FUNCTION_BLOCK Robotino (* Basic Function Block Type *)
  (* Standard: 61499-2 *)
  (* Version 0.0, 18/10/2022, Pranay Jhunjhunwala, Schneider Electric, Template *)
  PACKAGE Main;
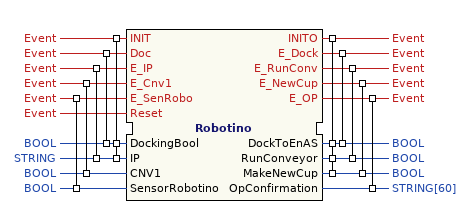
  EVENT_INPUT
    INIT WITH DockingBool, IP; (* Initialization Request *)
    Doc WITH DockingBool; (* Normal Execution Request *)
    E_IP WITH IP;
    E_Cnv1 WITH CNV1;
    E_SenRobo WITH SensorRobotino;
    Reset;
  END_EVENT
  EVENT_OUTPUT
    INITO WITH DockToEnAS, RunConveyor, MakeNewCup; (* Initialization Confirm *)
    E_Dock WITH DockToEnAS; (* Execution Confirmation *)
    E_RunConv WITH RunConveyor;
    E_NewCup WITH MakeNewCup;
    E_OP WITH OpConfirmation;
  END_EVENT
  VAR_INPUT
    DockingBool : BOOL; (* Input event qualifier *)
    IP : STRING;
    CNV1 : BOOL;
    SensorRobotino : BOOL;
  END_VAR
  VAR_OUTPUT
    DockToEnAS : BOOL; (* Output event qualifier *)
    RunConveyor : BOOL;
    MakeNewCup : BOOL;
    OpConfirmation : STRING[60];
  END_VAR
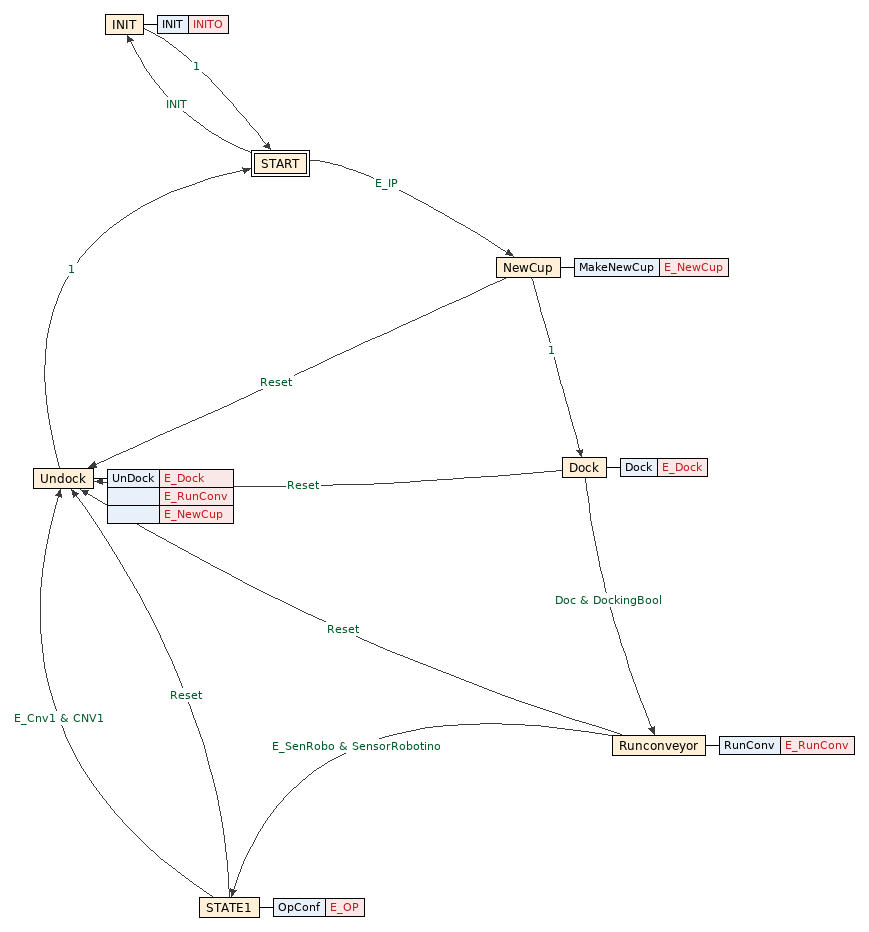
  EC_STATES
    START; (* Initial State *)
    INIT : INIT -> INITO; (* Initialization *)
    NewCup : MakeNewCup -> E_NewCup;
    Dock : Dock -> E_Dock;
    Runconveyor : RunConv -> E_RunConv;
    Undock : UnDock -> E_Dock, -> E_RunConv, -> E_NewCup;
    STATE1 : OpConf -> E_OP;
  END_STATES
  EC_TRANSITIONS
    START TO INIT := INIT;
    INIT TO START := 1;
    START TO NewCup := E_IP;
    NewCup TO Dock := 1;
    Dock TO Runconveyor := Doc & DockingBool;
    STATE1 TO Undock := E_Cnv1 & CNV1;
    Undock TO START := 1;
    NewCup TO Undock := Reset;
    Dock TO Undock := Reset;
    Runconveyor TO Undock := Reset;
    Runconveyor TO STATE1 := E_SenRobo & SensorRobotino;
    STATE1 TO Undock := Reset;
  END_TRANSITIONS
  ALGORITHM INIT IN ST: (* Initialization algorithm *)
;
  END_ALGORITHM
  ALGORITHM MakeNewCup IN ST: (* Normally executed algorithm *)
MakeNewCup := TRUE;
  END_ALGORITHM
  ALGORITHM Dock IN ST:
DockToEnAS := TRUE;
  END_ALGORITHM
  ALGORITHM RunConv IN ST:
RunConveyor := TRUE;
  END_ALGORITHM
  ALGORITHM UnDock IN ST:
DockToEnAS := FALSE;
RunConveyor := FALSE;
MakeNewCup := FALSE;
  END_ALGORITHM
  ALGORITHM OpConf IN ST:
OpConfirmation := 'R_DONE';
  END_ALGORITHM
END_FUNCTION_BLOCK
